// TIA Portal V19 export
TYPE "LEXCHANGETRAY_typeLogistics_interface"
// stored: Access Published
   STRUCT
      init : Bool;
      deliver : "LEXCHANGETRAY_typeLogistics_deliver_interface";
      recieve : "LEXCHANGETRAY_typeLogistics_recieve_interface";
   END_STRUCT;
END_TYPE
